{attribute 'GeneratedUsingTerminal: EL2521-0000-1016'}
{attribute addProperty BoxType "EL2521-0000-1016"}
{attribute addProperty Id "Target_counter_valueAT %Q*UINT2"}
{attribute addProperty CRC "1547018109"}
{attribute addProperty Size "2"}
TYPE PTO_Target_compact_5C359F7D :
STRUCT
	{attribute addProperty Name "Target_counter_value"}
	Target_counter_value AT %Q* : UINT;
END_STRUCT
END_TYPE

(* stored: Version 1.2.0.0, ProductVersion 3.1.4024.9
   DUT PTO_Target_compact_5C359F7D: Id {49b8a453-936f-4175-bee4-af2a01abc7bd} *)
